// General interface for error classes.
INTERFACE FsI_Error EXTENDS FsI_Unknown

PROPERTY Code : FsT_ErrCode
GET
END_GET
END_PROPERTY

PROPERTY Message : FsT_ErrMsg
GET
END_GET
END_PROPERTY

END_INTERFACE

(* stored: Version 1.1.0.1, ProductVersion 3.1.4024.4
   Itf FsI_Error: Id {8e2b39cc-44a5-4e58-81fd-0af79ce0a762}
   Folder Properties: Id {7c2e6905-3f51-4d36-9212-519664214bc2}
   Property Code: Id {46e2eaad-514a-48b2-ba14-98e93fdcaa6e}
   Get Get: Id {d1db998b-1f76-4d66-b62b-b99c1658358e}
   Property Message: Id {5984187f-15d0-4cc5-8716-8d1d9ccfc646}
   Get Get: Id {37ebe30e-d19b-4e5c-98da-6ac553ccdea0} *)
